// TIA Portal V14 SP1 export
// export: Created 2019-04-23T05:55:15.4382654Z, ExportSetting WithDefaults, WithReadOnly, DisplayName Totally Integrated Automation Portal, DisplayVersion V14 SP1 Update 6, DisplayName TIA Portal Openness, DisplayVersion V14 SP1 Update 6, DisplayName STEP 7 Professional, DisplayVersion V14 SP1 Update 6, DisplayName WinCC Professional, DisplayVersion V14 SP1 Update 6
FUNCTION_BLOCK "VBV2_Vibrating_screen_Cleaning_1"   // FB2010, LAD
TITLE = Управление автоочисткой вибросита / Управление очисткой вибросита
{ S7_Optimized_Access := 'FALSE' }
VERSION : 0.1
// stored: AutoNumber false, CodeModifiedDate 2019-03-07T08:39:59.0703225Z, CompileDate 2019-03-07T08:39:59.0857315Z, CreationDate 2019-02-26T05:18:41.6523018Z, InterfaceModifiedDate 2018-05-22T07:48:13.1874699Z, IsConsistent true, IsIECCheckEnabled false, IsKnowHowProtected false, ISMultiInstanceCapable true, IsWriteProtected false, LibraryConformanceStatus Warning: The block contains direct access to inputs, outputs, bit memories, indirect access to the registry or indirect access to external memory areas that are unknown at the time of compilation., ModifiedDate 2019-03-07T08:39:59.0703225Z, ParameterModified 2017-07-09T13:16:10.9043445Z, StructureModified 2018-05-11T05:29:45.0609697Z, UDAEnableTagReadback false
   VAR DB_SPECIFIC
      HMI : Struct
         CMD : Struct
            ON_Auto_Clean : Bool := true;   // Разрешение режима автооочистки вибросита
            Spare : Bool;
            Spare_1 : Bool;
            Spare_2 : Bool;
            Spare_3 : Bool;
            Spare_4 : Bool;
            Spare_5 : Bool;
            Spare_6 : Bool;
         END_STRUCT;
         DATA : Struct
            StatusWork : Int;   // Режим работы
            WorkTIme_sec : Int := 600;   // Заданное время работы перед очисткой
            CleanTIme_sec : Int := 40;   // Заданное время очистки вибросита
            WorkTime_Counter : Int;   // Время работа вибросита / Время работы вибросита
            CleanTime_Counter : Int;   // Время очистки вибросита
         END_STRUCT;
      END_STRUCT;
      Off_Time : Time;
      Cleaning_Request : Bool;   // 1 - необходимость очистки
      Spare : Bool;
      Spare_1 : Bool;
      Spare_2 : Bool;
      Spare_3 : Bool;
      Spare_4 : Bool;
      Spare_5 : Bool;
      Spare_6 : Bool;
   END_VAR
   VAR_TEMP
      Timer_ET : Time;
      StopTime : Time;
      Temp_BIT : Bool;
   END_VAR
   VAR_TEMP   // added for the SCL form of the ladder/FBD networks
      _w1 : Bool;
   END_VAR
BEGIN

REGION Network 1: Блок активирования очередной очистки вибросита после истечения счетчика его работы
END_REGION

REGION Network 2: Счетчик работы во время загрузки продукта
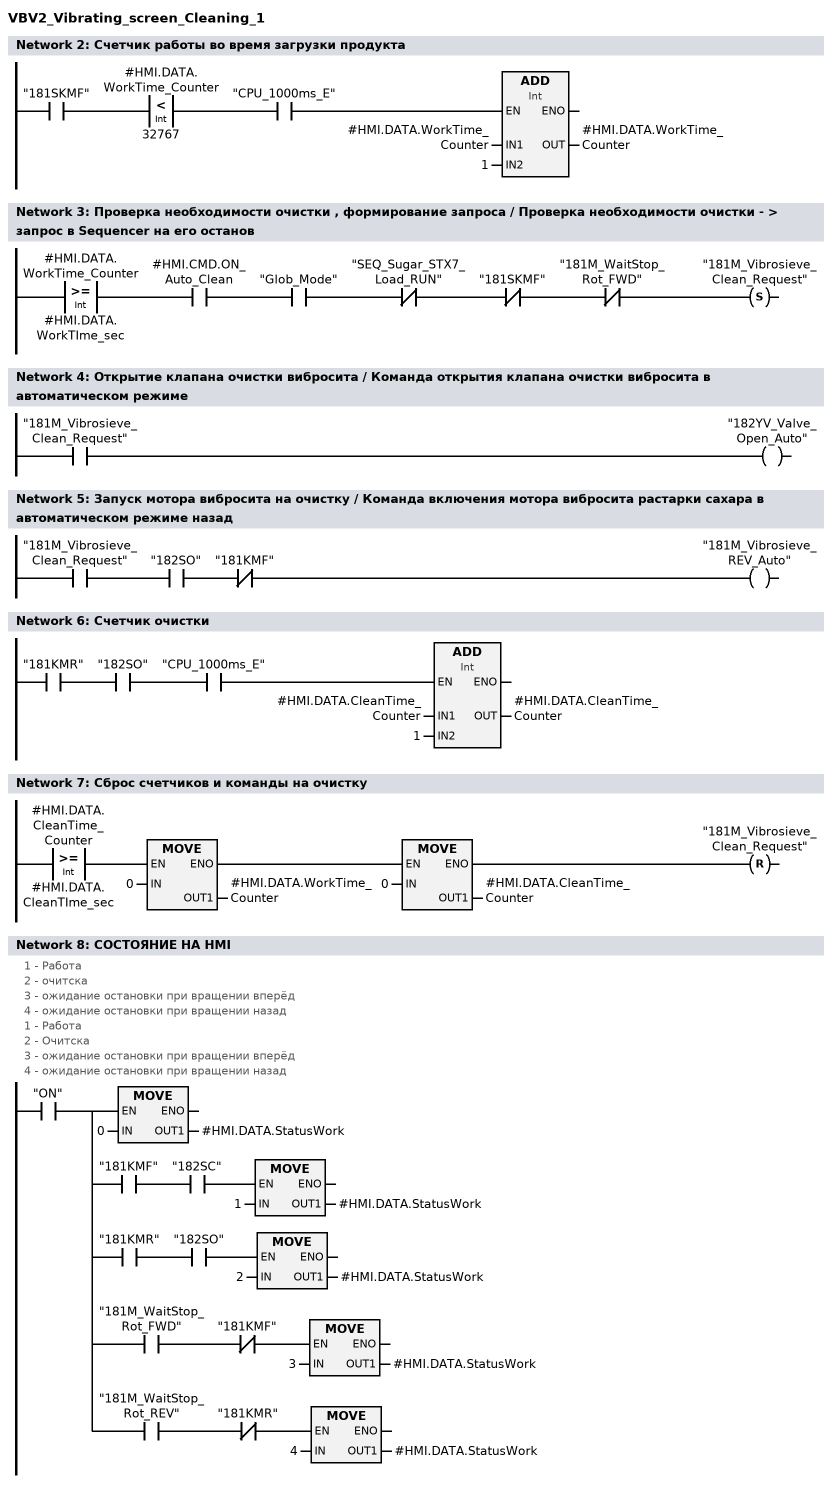
   RUNG wire#powerrail
      Contact( "181SKMF" )
      { S7_Templates := "SrcType := Int" } LT_Contact(in1 := #HMI.DATA.WorkTime_Counter, in2 := 32767)
      Contact( "CPU_1000ms_E" )
      { S7_Templates := "SrcType := Int"; S7_GenerateENO := "TRUE" } Add(in1 := #HMI.DATA.WorkTime_Counter, in2 := 1, out => #HMI.DATA.WorkTime_Counter)
   END_RUNG
   // the same network as SCL:
   IF "181SKMF" AND (#HMI.DATA.WorkTime_Counter < 32767) AND "CPU_1000ms_E" THEN
       #HMI.DATA.WorkTime_Counter := #HMI.DATA.WorkTime_Counter + 1;
   END_IF;
END_REGION

REGION Network 3: Проверка необходимости очистки , формирование запроса / Проверка необходимости очистки - > запрос в Sequencer на его останов
   RUNG wire#powerrail
      { S7_Templates := "SrcType := Int" } GE_Contact(in1 := #HMI.DATA.WorkTime_Counter, in2 := #HMI.DATA.WorkTIme_sec)
      Contact( #HMI.CMD.ON_Auto_Clean )
      Contact( "Glob_Mode" )
      I_Contact( "SEQ_Sugar_STX7_Load_RUN" )
      I_Contact( "181SKMF" )
      I_Contact( "181M_WaitStop_Rot_FWD" )
      S_Coil( "181M_Vibrosieve_Clean_Request" )
   END_RUNG
   // the same network as SCL:
   IF (#HMI.DATA.WorkTime_Counter >= #HMI.DATA.WorkTIme_sec) AND #HMI.CMD.ON_Auto_Clean AND "Glob_Mode" AND NOT "SEQ_Sugar_STX7_Load_RUN" AND NOT "181SKMF" AND NOT "181M_WaitStop_Rot_FWD" THEN
       "181M_Vibrosieve_Clean_Request" := TRUE;
   END_IF;
END_REGION

REGION Network 4: Открытие клапана очистки вибросита / Команда открытия клапана очистки вибросита в автоматическом режиме
   RUNG wire#powerrail
      Contact( "181M_Vibrosieve_Clean_Request" )
      Coil( "182YV_Valve_Open_Auto" )
   END_RUNG
   // the same network as SCL:
   "182YV_Valve_Open_Auto" := "181M_Vibrosieve_Clean_Request";
END_REGION

REGION Network 5: Запуск мотора вибросита на очистку / Команда включения мотора вибросита растарки сахара в автоматическом режиме назад
   RUNG wire#powerrail
      Contact( "181M_Vibrosieve_Clean_Request" )
      Contact( "182SO" )
      I_Contact( "181KMF" )
      Coil( "181M_Vibrosieve_REV_Auto" )
   END_RUNG
   // the same network as SCL:
   "181M_Vibrosieve_REV_Auto" := "181M_Vibrosieve_Clean_Request" AND "182SO" AND NOT "181KMF";
END_REGION

REGION Network 6: Счетчик очистки
   RUNG wire#powerrail
      Contact( "181KMR" )
      Contact( "182SO" )
      Contact( "CPU_1000ms_E" )
      { S7_Templates := "SrcType := Int"; S7_GenerateENO := "TRUE" } Add(in1 := #HMI.DATA.CleanTime_Counter, in2 := 1, out => #HMI.DATA.CleanTime_Counter)
   END_RUNG
   // the same network as SCL:
   IF "181KMR" AND "182SO" AND "CPU_1000ms_E" THEN
       #HMI.DATA.CleanTime_Counter := #HMI.DATA.CleanTime_Counter + 1;
   END_IF;
END_REGION

REGION Network 7: Сброс счетчиков и команды на очистку
   RUNG wire#powerrail
      { S7_Templates := "SrcType := Int" } GE_Contact(in1 := #HMI.DATA.CleanTime_Counter, in2 := #HMI.DATA.CleanTIme_sec)
      { S7_GenerateENO := "TRUE" } Move(in := 0, out1 => #HMI.DATA.WorkTime_Counter)
      { S7_GenerateENO := "TRUE" } Move(in := 0, out1 => #HMI.DATA.CleanTime_Counter)
      R_Coil( "181M_Vibrosieve_Clean_Request" )
   END_RUNG
   // the same network as SCL:
   // ENO of a box is taken as its EN; it also drops when the box reports an error
   IF #HMI.DATA.CleanTime_Counter >= #HMI.DATA.CleanTIme_sec THEN #HMI.DATA.WorkTime_Counter := 0; END_IF;
   #_w1 := #HMI.DATA.CleanTime_Counter >= #HMI.DATA.CleanTIme_sec;
   IF #_w1 THEN
       #HMI.DATA.CleanTime_Counter := 0;
       "181M_Vibrosieve_Clean_Request" := FALSE;
   END_IF;
END_REGION

REGION Network 8: СОСТОЯНИЕ НА HMI
   // 1 - Работа
   // 2 - очитска
   // 3 - ожидание остановки при вращении вперёд
   // 4 - ожидание остановки при вращении назад
   // 1 - Работа
   // 2 - Очитска
   // 3 - ожидание остановки при вращении вперёд
   // 4 - ожидание остановки при вращении назад
   RUNG wire#powerrail
      Contact( "ON" )
      wire#w1
      { S7_GenerateENO := "TRUE" } Move(in := 0, out1 => #HMI.DATA.StatusWork)
   END_RUNG
   RUNG wire#w1
      Contact( "181KMF" )
      Contact( "182SC" )
      { S7_GenerateENO := "TRUE" } Move(in := 1, out1 => #HMI.DATA.StatusWork)
   END_RUNG
   RUNG wire#w1
      Contact( "181KMR" )
      Contact( "182SO" )
      { S7_GenerateENO := "TRUE" } Move(in := 2, out1 => #HMI.DATA.StatusWork)
   END_RUNG
   RUNG wire#w1
      Contact( "181M_WaitStop_Rot_FWD" )
      I_Contact( "181KMF" )
      { S7_GenerateENO := "TRUE" } Move(in := 3, out1 => #HMI.DATA.StatusWork)
   END_RUNG
   RUNG wire#w1
      Contact( "181M_WaitStop_Rot_REV" )
      I_Contact( "181KMR" )
      { S7_GenerateENO := "TRUE" } Move(in := 4, out1 => #HMI.DATA.StatusWork)
   END_RUNG
   // the same network as SCL:
   IF "ON" THEN #HMI.DATA.StatusWork := 0; END_IF;
   IF "ON" AND "181KMF" AND "182SC" THEN #HMI.DATA.StatusWork := 1; END_IF;
   IF "ON" AND "181KMR" AND "182SO" THEN #HMI.DATA.StatusWork := 2; END_IF;
   IF "ON" AND "181M_WaitStop_Rot_FWD" AND NOT "181KMF" THEN #HMI.DATA.StatusWork := 3; END_IF;
   IF "ON" AND "181M_WaitStop_Rot_REV" AND NOT "181KMR" THEN #HMI.DATA.StatusWork := 4; END_IF;
END_REGION

NETWORK
TITLE = end
      SET;
      SAVE;

END_FUNCTION_BLOCK
